// TIA Portal V15.1 export
// export: Created 2024-06-21T08:41:08.8538239Z, ExportSetting WithDefaults, DisplayName Totally Integrated Automation Portal, DisplayVersion V15.1 Update 5, DisplayName TIA Portal Openness, DisplayVersion V15.1 Update 5, DisplayName SINAMICS Startdrive Advanced, DisplayVersion V15.1, DisplayName G130, G150, S120, S150, SINAMICS MV, S210, DisplayVersion V15.1, DisplayName G110M, G120, G120C, G120D, G120P, DisplayVersion V15.1, DisplayName STEP 7 Professional, DisplayVersion V15.1 Update 5, DisplayName STEP 7 Safety, DisplayVersion V15.1, DisplayName WinCC Professional, DisplayVersion V15.1 Update 5, DisplayName SIMATIC Visualization Architect, DisplayVersion V15.1
FUNCTION "LGBProdSpeed-Config" : Void   // FC6699, FBD
TITLE = LGBProdSpeed-Config
{ S7_Optimized_Access := 'TRUE' }
VERSION : 0.1
// stored: AutoNumber false, IsIECCheckEnabled false, SetENOAutomatically False, UDAEnableTagReadback false
   VAR_INPUT
      C_SetpointsFromCR : Bool;   // Setpoint from control room are used
      "C_Btn50%" : Bool;   // Button 50% production speed is visible on HMI
      C_LowestCycleTime : Int;   // Lowest cycle time in sec
      C_HighestCycleTime : Int;   // Highest cycle time in sec
   END_VAR
   VAR_IN_OUT
      IO_Config : "ProdSpeedConfig";   // Config
   END_VAR
BEGIN

REGION Network 1: **** 1 Inputs **** Config
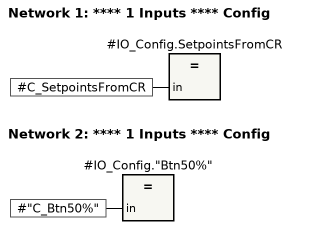
   #IO_Config.SetpointsFromCR := #C_SetpointsFromCR;
END_REGION

REGION Network 2: **** 1 Inputs **** Config
   #IO_Config."Btn50%" := #"C_Btn50%";
END_REGION

NETWORK
TITLE = **** 1 Inputs **** Move Config UDT
// Move Config
      L     #C_LowestCycleTime;
      T     #IO_Config.LowestCycleTime;
      L     #C_HighestCycleTime;
      T     #IO_Config.HighestCycleTime;
END_FUNCTION
